{attribute 'no_explicit_call' := 'do not call this POU directly'}
FUNCTION_BLOCK PUBLIC FINAL FB_TcUnitAdapter IMPLEMENTS I_TestFrameWorkAdapter
VAR
	fbVerify : FB_Snappy;
	eStep : (INIT, VERIFYING, GET_RESULT, FINISHED) := INIT;
END_VAR

PROPERTY sTestName : REFERENCE TO T_MaxString
GET
sTestName REF= GVL_TcUnit.CurrentTestNameBeingCalled;
END_GET
END_PROPERTY

PROPERTY sTestSuiteName : REFERENCE TO T_MaxString
GET
sTestSuiteName REF= GVL_TcUnit.CurrentTestSuiteBeingCalled^.InstancePath;
END_GET
END_PROPERTY

METHOD Verify : HRESULT
VAR_INPUT
	anyArg	: ANY;
END_VAR

VAR	
	hr : HRESULT;
	pTestSuite : POINTER TO FB_TestSuite;
END_VAR
pTestSuite := GVL_TcUnit.CurrentTestSuiteBeingCalled;

IF pTestSuite = NULL THEN
	Verify := Tc2_System.E_HRESULTAdsErr.INVALIDCONTEXT;
	RETURN;
END_IF

CASE eStep OF

	INIT:		
		hr := fbVerify.Configure().UseDefaults().UseTestFramework(THIS^).Build();
		IF SUCCEEDED(hr) THEN
			eStep := VERIFYING;
			hr := S_PENDING;
		ELSE
			pTestSuite^.AssertEquals_DINT(Expected:= S_OK,
								Actual:= hr,
								Message:= 'Configuration failed');			
			eStep := FINISHED;
		END_IF

	VERIFYING:
		hr := fbVerify.Verify(anyArg:= anyArg);
		IF SUCCEEDED_AND_NOT_PENDING(hr)THEN
			eStep := GET_RESULT;
			hr := S_PENDING;
		ELSIF FAILED(hr) AND hr = E_HESULT_AdsErr.ERR_TARGETPORTNOTFOUND THEN
			pTestSuite^.AssertEquals_DINT(Expected:= S_OK,
							Actual:= hr,
							Message:= 'Targetport not found! Make sure, TcHaxx.Snappy.CLI is running, and a ADS route has been established.');
		ELSIF FAILED(hr) THEN
			pTestSuite^.AssertEquals_DINT(Expected:= S_OK,
							Actual:= hr,
							Message:= 'One or more errors occured');
			eStep := FINISHED;
		END_IF

	GET_RESULT:
		hr := fbVerify.stVerificationResult.hr;
		IF FAILED(hr) THEN
				pTestSuite^.AssertEquals_DINT(Expected:= S_OK,
								Actual:= hr,
								Message:= fbVerify.stVerificationResult.sDiff);
		END_IF;
		eStep := FINISHED;

	FINISHED:
		eStep := INIT;
END_CASE

Verify := hr;
END_METHOD

END_FUNCTION_BLOCK

(* stored: Version 1.1.0.1, ProductVersion 3.1.4026.18
   POU FB_TcUnitAdapter: Id {9a3e8679-ffe2-40a8-b498-cb88fd65cd9f}, SpecialFunc None
   Property sTestName: Id {41f90fb1-f99e-48f8-ac93-773cef804bd1}
   Get Get: Id {991bd039-c0a6-42b0-88dc-c080ece7ad5f}
   Property sTestSuiteName: Id {121e7dc6-f84b-4ea6-bc0f-fdcd5cae0dcc}
   Get Get: Id {9529d8ca-ea0b-4332-bbe6-758860146803}
   Method Verify: Id {814f1f18-1621-4841-9501-0e71bbfe79a4} *)
